// TwinCAT 3 PLC project Library
// Title: lcls-twincat-rail
// Company: SLAC
// ProjectVersion: 0.0.0
// ProgramVersion: 3.1.4022.7
// libraries:
//   Tc2_EtherCAT, * (Beckhoff Automation GmbH)
//   Tc2_Standard, * (Beckhoff Automation GmbH)
//   Tc2_System, * (Beckhoff Automation GmbH)
//   Tc3_Module, * (Beckhoff Automation GmbH)
// project tree:
//   DUTs/ DUT_70x1CoeData.TcDUT, E_CoeState.TcDUT
//   GVLs/ GVL_COE.TcGVL
//   / PlcTask.TcTTO
//   POUs/ FB_Read70x1CoeData.TcPOU, MAIN.TcPOU
//   Utils/ FB_FindSecondaryAddr.TcPOU
// real-time tasks:
//   TASK PlcTask: cycle T#10ms, priority 20, ADS port 350

CONFIGURATION Library
    RESOURCE PLC ON TwinCAT3
        TASK PlcTask(INTERVAL := T#10ms, PRIORITY := 20);
        PROGRAM MAIN WITH PlcTask : MAIN;
    END_RESOURCE
END_CONFIGURATION

// ---- DUTs/DUT_70x1CoeData.TcDUT
TYPE DUT_70x1CoeData :
STRUCT
     (* Hardware *)
    //Readbacks
    {attribute 'pytmc' := '
     pv: TRM:NAME
     io: i
     field: DESC beck terminal type
    '}
    sDeviceName : STRING(35);
    {attribute 'pytmc' := '
     pv: MAX:CUR
     io: i
     field: DESC Max Current
    '}
    nMaxCurrent : WORD;
    {attribute 'pytmc' := '
     pv: REDUC:CUR
     io: i
     field: DESC Reduced Current
    '}
    nReducedCurrent : WORD;
    {attribute 'pytmc' := '
     pv: NOM:VOL
     io: i
     field: DESC Nominal Voltage
    '}
    nNominalVoltage: WORD;
    {attribute 'pytmc' := '
     pv: MTR:STP
     io: i
     field: DESC Motor Fullsteps
    '}
    nMotorFullSteps: WORD;
    {attribute 'pytmc' := '
     pv: SPD:RNG
     io: i
     field: DESC Speed Range
    '}
    nSpeedRange: WORD;
END_STRUCT
END_TYPE

// ---- DUTs/E_CoeState.TcDUT
{attribute 'qualified_only'}
TYPE E_CoeState :
(
    Init := 0,
    Read,
    ReadPeriodically,
    Error,
    Idle,
    PreRead,
    Calculate
);
END_TYPE

// ---- GVLs/GVL_COE.TcGVL
{attribute 'qualified_only'}
VAR_GLOBAL
    CONSTANT
    EC_MAX_SECONDARY :  BYTE := 10;
    MAX_STRING_SIZE : BYTE := 81;
    NUM_70x1_COE_PARAM : BYTE := 6;
    NUM_SUP_70x1 : BYTE := 4;
END_VAR

// ---- POUs/MAIN.TcPOU
PROGRAM MAIN
VAR
END_VAR

END_PROGRAM

// ---- POUs/FB_Read70x1CoeData.TcPOU
FUNCTION_BLOCK FB_Read70x1CoeData
VAR_INPUT
   userNetId             : T_AmsNetId := ''; // Have to be entered
END_VAR
VAR_OUTPUT
    {attribute 'pytmc' := '
        pv: COE
    '}
    aCoeData : ARRAY[0..9] OF DUT_70x1CoeData;
    userSlaveAddr         : POINTER TO UINT;
END_VAR
VAR_IN_OUT
END_VAR
VAR
   fbCoeRead           : FB_EcCoESdoRead;  // Function Block for reading from CoE
   fbGetSecondaries   : FB_FindSecondaryAddr;  // Function Block for reading Secondary Addresses

   nNumCoeParam           : BYTE := GVL_COE.NUM_70x1_COE_PARAM;
   bInit               : BOOL := TRUE;  // Kicks off Secondary Address read.
   // NEED TO MANUALLY UPDATE GVL_COE SIZES
   aCoeIndex           : ARRAY[0..GVL_COE.NUM_70x1_COE_PARAM - 1] OF BYTE := [0, 1, 2, 3, 6, 5];
   aCoeAddr            : ARRAY[0..GVL_COE.NUM_70x1_COE_PARAM - 1] OF WORD :=   [16#1008, 16#8010, 16#8010, 16#8010, 16#8010, 16#8012];
   aTerminalType       : ARRAY[0..GVL_COE.NUM_SUP_70x1] OF STRING := ['EL7031', 'EL7041', 'EL7041-1000', 'EL7047'];
   {attribute 'pytmc' := '
        pv: READ
        io: io
   '}
   bStartRead             : BOOL := FALSE;    // Sign for start reading CoE
   eState   			: E_CoeState := E_CoeState.Init;
   nReadIndex           : BYTE :=  0;
   nSecondaryIndex          : BYTE := 0;
   nSecondaries              : UINT := 0;
   pDstBuf              :   POINTER TO WORD;
   cbBufLen   : UDINT;

   bValidTerm : BOOL;
   nForLoop : INT;

END_VAR

CASE eState OF
E_CoeState.Init:
   fbGetSecondaries(userNetId:=userNetId, bExecute:= bInit);
   bInit := FALSE;
//Needs Error Checking
   IF NOT fbGetSecondaries.bBusy THEN
        userSlaveAddr := ADR(fbGetSecondaries.userSlaveAddr);
        nSecondaries := fbGetSecondaries.nSecondaries;
        eState := E_CoeState.PreRead;// Next state for reading
   END_IF
E_CoeState.PreRead:
   IF bStartRead THEN
      eState := E_CoeState.Read;// Next state for reading
      fbCoeRead(bExecute := FALSE);// Prepare CoE-Access: Read an object/ sub index
      bStartRead := FALSE;
   END_IF
;

E_CoeState.Read:

     CASE nReadIndex OF
       0:
         pDstBuf := ADR(aCoeData[nSecondaryIndex].sDeviceName);
       1:
         pDstBuf := ADR(aCoeData[nSecondaryIndex].nMaxCurrent);
       2:
         pDstBuf := ADR(aCoeData[nSecondaryIndex].nReducedCurrent);
       3:
         pDstBuf := ADR(aCoeData[nSecondaryIndex].nNominalVoltage);
       4:
         pDstBuf := ADR(aCoeData[nSecondaryIndex].nMotorFullSteps);
       5:
         pDstBuf := ADR(aCoeData[nSecondaryIndex].nSpeedRange);

     END_CASE
    IF nReadIndex = 0 THEN
    cbBufLen := GVL_COE.MAX_STRING_SIZE;
    ELSE
    cbBufLen := SIZEOF(pDstBuf^);
    END_IF
   // Read entry
   fbCoeRead(
   sNetId:= userNetId,
   nSlaveAddr:= userSlaveAddr[nSecondaryIndex],
   nSubIndex:= aCoeIndex[nReadIndex],
   nIndex:= aCoeAddr[nReadIndex],
   pDstBuf:= pDstBuf,
   cbBufLen:= cbBufLen,
   bExecute:= TRUE,
   tTimeout:= T#1S
   );
   eState := E_CoeState.Idle; // Next state
E_CoeState.Idle:
   fbCoeRead();        // Execute CoE read until done
   IF fbCoeRead.bError THEN
      eState := E_CoeState.Error;     // Error case
   ELSE
      IF NOT fbCoeRead.bBusy THEN
             eState := E_CoeState.PreRead;
             IF nReadIndex = 0 THEN
                // Make sure its an EL70x1
                bValidTerm := FALSE;
                FOR nForLoop := 0 TO GVL_COE.NUM_SUP_70x1 - 1 DO
                    IF aCoeData[nSecondaryIndex].sDeviceName = aTerminalType[nForLoop] THEN
                        bValidTerm := TRUE;
                        EXIT;
                    END_IF
                END_FOR
                IF bValidTerm THEN
                    // Valid terminal, keep reading
                    bStartRead := TRUE;
                    nReadIndex := nReadIndex + 1;
                ELSIF nSecondaryIndex < nSecondaries - 1 THEN
                    // Invalid terminal, looks for next temrinal
                    nSecondaryIndex := nSecondaryIndex + 1;
                    nReadIndex := 0;
                    //estate := E_CoeState.Init;
                    estate := E_CoeState.PreRead;
                    bStartRead := TRUE;
                ELSE
                    //Invalid terminal and none left.
                    //Done reading, reset indices
                    nReadIndex := 0;
                    nSecondaryIndex := 0;
                END_IF

             ELSIF nReadIndex < nNumCoeParam - 1 THEN
                bStartRead := TRUE;
                nReadIndex := nReadIndex + 1;
             ELSIF nReadIndex = nNumCoeParam - 1 AND nSecondaryIndex < nSecondaries - 1 THEN
                nReadIndex := 0;
                nSecondaryIndex := nSecondaryIndex + 1;
                bStartRead := TRUE;
             ELSE
                //Done reading, reset indices
                nReadIndex := 0;
                nSecondaryIndex := 0;
                ;
             END_IF
         END_IF
   END_IF
E_CoeState.Error:
    IF fbCoeRead.nErrId = 13
        //ERR_PORTNOTCONNECTED wasnt supported, non CoE Terminal.
     OR fbCoeRead.nErrId = 1797
        //ADSERR_DEVICE_INVALIDOFFSET, not an EL70x1
     OR fbCoeRead.nErrId = 1795 THEN
        //ADSERR_DEVICE_INVALIDSIZE, not an EL70x1
        IF nSecondaryIndex < nSecondaries - 1 THEN
            nSecondaryIndex := nSecondaryIndex + 1;
            nReadIndex := 0;
            estate := E_CoeState.PreRead;
            bStartRead := TRUE;
        END_IF
    END_IF
END_CASE

END_FUNCTION_BLOCK

// ---- Utils/FB_FindSecondaryAddr.TcPOU
FUNCTION_BLOCK FB_FindSecondaryAddr
VAR_INPUT
    userNetId             : T_AmsNetId := ''; // Have to be entered
    bExecute                : BOOL;
END_VAR
VAR_OUTPUT
    userSlaveAddr         : ARRAY[0..GVL_COE.EC_MAX_SECONDARY] OF UINT;
    nSecondaries           : UINT := 0;
    bBusy              : BOOL := FALSE;
END_VAR
VAR
    fbGetSecondary : FB_EcGetAllSlaveAddr;
    eState   			: E_CoeState := E_CoeState.Init;
END_VAR

CASE eState OF
E_CoeState.Init:
    IF bExecute THEN
        bBusy := TRUE;
        eState := E_CoeState.Read;
        bExecute := FALSE;
    END_IF
E_CoeState.Read:
    fbGetSecondary(
        sNetId:=userNetId,
        pAddrBuf:=ADR(userSlaveAddr),
        cbBufLen:=SIZEOF(userSlaveAddr),
        bExecute := TRUE,
    );
    eState := E_CoeState.Idle;

E_CoeState.Idle:
    IF fbGetSecondary.bError THEN
        eState := E_CoeState.Error;
    ELSE
        IF NOT fbGetSecondary.bBusy THEN
            eState := E_CoeState.Init;
            bBusy := FALSE;
            nSecondaries := fbGetSecondary.nSlaves;
        ELSE
            fbGetSecondary(
                sNetId:=userNetId,
                pAddrBuf:=ADR(userSlaveAddr),
                cbBufLen:=SIZEOF(userSlaveAddr),
                bExecute := FALSE );
        END_IF
    END_IF
E_CoeState.Error:
;
END_CASE

END_FUNCTION_BLOCK
